PROGRAM MAIN
VAR
		bStart  :BOOL;
		bEnable :BOOL;
		nINT : INT := -32768;
	    nUINT : UINT := 65535;
	    fREAL : REAL := 255.255;
		sPowerStatus: STRING := 'Power Off'; 
		nFloatConversion:INT;
		fFloatConversion:LREAL;
END_VAR

bEnable:= bStart;
fFloatConversion:=INT_TO_LREAL(nFloatConversion);

END_PROGRAM

(* stored: Version 1.1.0.1, ProductVersion 3.1.4024.12
   POU MAIN: Id {1d13e196-1409-403d-8338-8ffee01bfd7d}, SpecialFunc None *)
